(*
SPDX-FileCopyrightText: © 2026 Oleksandr Tiutyk <trofimich@gmail.com>
SPDX-License-Identifier: MIT
License: https://opensource.org/license/mit
*)

INTERFACE ISystemException EXTENDS IException

{attribute 'monitoring' := 'call'}
PROPERTY ExceptionCode : __SYSTEM.ExceptionCode
GET
END_GET
END_PROPERTY

END_INTERFACE

(* stored: Version 1.1.0.1
   Itf ISystemException: Id {7870ea65-b79e-4a5f-a0cf-37b06b88ed45}
   Property ExceptionCode: Id {15970fe0-8365-4901-b4a4-73314108321e}
   Get Get: Id {5aed6761-fded-45fb-a3b9-33b86ea1a435} *)
